// TIA Portal V16 export
// export: Created 2024-12-03T15:41:45.9905796Z, ExportSetting WithReadOnly, DisplayName Totally Integrated Automation Portal, DisplayVersion V16 Update 6, DisplayName TIA Portal Version Control Interface, DisplayVersion V16 Update 2, DisplayName TIA Portal Openness, DisplayVersion V16 Update 6, DisplayName TIA Portal Teamcenter Gateway, DisplayVersion V16, DisplayName SINAMICS Startdrive Advanced, DisplayVersion V16 Update 5, DisplayName SINAMICS Startdrive G130, G150, S120, S150, SINAMICS MV, S210, DisplayVersion V16 Update 5, DisplayName SINAMICS Startdrive G110M, G120, G120C, G120D, G120P, G115D, DisplayVersion V16 Update 5, DisplayName STEP 7 Professional, DisplayVersion V16 Update 6, DisplayName STEP 7 Safety, DisplayVersion V16, DisplayName WinCC Advanced / Unified PC, DisplayVersion V16 Update 6
TYPE "Conveyor_UDT"
// stored: CreationDate 2021-07-13T07:41:36.2278727Z, InterfaceModifiedDate 2023-07-16T10:12:43.624232Z, IsConsistent true, LibraryConformanceStatus The object is library-conformant., ModifiedDate 2023-07-16T10:12:43.624232Z
   STRUCT
      Settings : Struct
         Mode { S7_SetPoint := 'True'} : Int;   // 0 ZPA MODE | 1 Buffer Mode | 2 Run till end mode
         AutomaticBuffering { S7_SetPoint := 'True'} : Bool := FALSE;   // Automatically switch between buffer mode and run till end mode if setting is run till end mode
         Direction { S7_SetPoint := 'True'} : Bool := FALSE;   // The normal direction of the conveyor
         EnergySave { S7_SetPoint := 'True'} : Bool := true;   // Save energy in run till end mode
         RunIddle { S7_SetPoint := 'True'} : Bool := false;
         AutoReset { S7_SetPoint := 'True'} : Bool := true;   // Auto reset conveyor when object is removed
         SentHoldOnCheckReceive { S7_SetPoint := 'True'} : Bool := false;   // OnlyRun conveyor during sent hold on when downstream is ready
         Timings { S7_SetPoint := 'True'} : "ConveyorTimes_UDT";
         Speed : Struct
            speed { S7_SetPoint := 'True'} : Real := 75.0;   // the speed in %
            UpstreamGain { S7_SetPoint := 'True'} : Real := 1.0;
            speedController { S7_SetPoint := 'True'} : Bool := FALSE;
         END_STRUCT;
         Alarms : Struct
            BlockDetectionOn { S7_SetPoint := 'True'} : Bool := true;
            BlockedAtStartSensor { S7_SetPoint := 'True'} : Bool;
            ParcelsToCloseDetectionOn { S7_SetPoint := 'True'} : Bool;
            ParcelsToLongDetectionOn { S7_SetPoint := 'True'} : Bool;
            ParcelToShortDetectionOn { S7_SetPoint := 'True'} : Bool;
            BlockRetrys { S7_SetPoint := 'True'} : Int := 1;
            SentTimeError { S7_SetPoint := 'True'} : Real := 3000.0;   // Also used for parcel to long detection
            TimeBetweenParcels { S7_SetPoint := 'True'} : Real := 500.0;   // Parcels to close detection
            MinSizeParcel { S7_SetPoint := 'True'} : Real := 100.0;
            MaxSizeParcel { S7_SetPoint := 'True'} : Real := 2200.0;
         END_STRUCT;
      END_STRUCT;
      Cmd : Struct
         Reset : Bool;
         ReInitialize : Bool;
         RunAuto : Bool;
         RunManual : Bool;
         SpeedAuto : Real;
         SpeedManual : Real;
         ReadyToReceive : Bool;
         ReadyToSent : Bool;
         InvertFlow : Bool;
         Direction : Bool;
         Accumulate : Struct
            Acc_ext_1 : Bool;
            Acc_ext_2 : Bool;
            Acc_ext_3 : Bool;
            Acc_ext_4 : Bool;
            Acc_ext_5 : Bool;
            Acc_TC_1 : Bool;
            Acc_TC_2 : Bool;
            Acc_TC_3 : Bool;
            Acc_Scan_1 : Bool;
            Acc_Scan_2 : Bool;
            Acc_Scan_3 : Bool;
            Acc_Scale_1 : Bool;
            Acc_Scale_2 : Bool;
            Acc_Scale_3 : Bool;
         END_STRUCT;
         StartRequestObject : Bool;
         StopRequestObject : Bool;
         IgnoreStandby : Bool;
         ManualOverride : Bool;
         Interlock : Bool;
      END_STRUCT;
      Input : Struct
         SensorStartHMI : Bool;
         SensorEndHMI : Bool;
         SensorAtStartLogic { S7_SetPoint := 'True'} : "SmartBooldt";
         SensorAtEndLogic { S7_SetPoint := 'True'} : "SmartBooldt";
         Running_FB : Bool;
         Interlock : Bool;
      END_STRUCT;
      Alarms : Struct
         BlockedReceive : "HmiAlarm";   // Conveyor is Blocked
         BlockedSending { S7_SetPoint := 'True'} : "HmiAlarm";
         ToClose { S7_SetPoint := 'True'} : "HmiAlarm";
         ToSmall { S7_SetPoint := 'True'} : "HmiAlarm";
         ToLong { S7_SetPoint := 'True'} : "HmiAlarm";
         MotorAlarm { S7_SetPoint := 'True'} : "HmiAlarm";
         AlarmActive { S7_SetPoint := 'True'} : "HmiAlarm";
         Status : Word;   // lsb : 0 blocked | 1 interlocked
      END_STRUCT;
      Status : Struct
         AccumulationOn : Bool;
         StartedAutoMode : Bool;
         ReadyForStandby : Bool;
         RequestForSending : Bool;
         ExecutingReceiveSequence : Bool;
         ExecutingSendingSequence : Bool;
         ObjectSentPulse : Bool;
         ObjectReceivePulse : Bool;
         GapTimeOk : Bool;
         Empty : Bool;
         ObjectOnConveyor : Bool;
         Initialized : Bool;
         ManualMode : Bool;
      END_STRUCT;
      TrackingCmd : Struct
         InductNewTracking : Bool;
         ClearTracking : Bool;
         NewTrackingId { S7_SetPoint := 'True'} : "Tracking_Simple_UDT_1";
      END_STRUCT;
      TrackingStat : Struct
         Current { S7_SetPoint := 'True'} : "Tracking_Simple_UDT_1";
         InSending { S7_SetPoint := 'True'} : "Tracking_Simple_UDT_1";
         TrackingReceived : Bool;
         TrackingCleared : Bool;
      END_STRUCT;
      Encoder { S7_SetPoint := 'True'} : "VirtualEncoder_UDT";
      DiagNostics : Struct
         ReceivedCounter : UDInt;
         SendingCounter : UDInt;
      END_STRUCT;
      Index { S7_SetPoint := 'True'} : Int;
      "Name" : String[25];
      Zone { S7_SetPoint := 'True'} : Int;
   END_STRUCT;
   // Settings.Timings.ConveyorLength := 2000.0;
   // Settings.Timings.InitDistance := 2000.0;
   // Settings.Timings.ReceiveDistance := 0.0;
   // Settings.Timings.SendDistance := 150.0;
   // Settings.Timings.SleepDistance := 1500.0;
   // Encoder.Settings.Base_M_min := 56.0;
END_TYPE
